// TIA Portal V20 export
FUNCTION "FillBuffers" : Void   // FC10050, SCL
TITLE = FillBuffers
{ S7_Optimized_Access := 'TRUE' }
AUTHOR : DIL
VERSION : 1.0
// stored: SetENOAutomatically false
   VAR_INPUT
      doneComRF160 : Bool;
      restartSync : Bool;
      epcId : Array[0..127] of Byte;
      data : Array[0..181] of Byte;
   END_VAR
   VAR_IN_OUT
      bufferIndex : Int;
      epcBuffer : Array[0..#MAXTAGCOUNT, 0..127] of Byte;
      dataBuffer : Array[0..#MAXTAGCOUNT, 0..181] of Byte;
   END_VAR
   VAR CONSTANT
      MAXTAGCOUNT : Int := 31;
   END_VAR
BEGIN
   //=============================================================================
   // Siemens AG
   // (c)Copyright (2022) All Rights Reserved
   //-----------------------------------------------------------------------------
   // Library: ---
   // Tested with: S7-1511-1 PN, FW V2.9
   // Engineering: TIA Portal V18 
   // Restrictions: ---
   // Requirements: ---
   // Functionality: Moves the data from the inputs to the InOuts when new data is available.
   // This FC was build to work with FB "ComRF160" and a buffer of size 32 for epcIds and datas.
   //-----------------------------------------------------------------------------
   // Change log table:
   // Version  Date       Expert in charge Changes applied
   // 01.00.00 01.09.2022 (User)           First released version
   //=============================================================================


   //===========================================================
   // Check for sync restart and reset buffers if necessary
   //===========================================================
   IF #doneComRF160 AND #restartSync THEN //make sure bufferIndex is in range of 0 to 31 to match buffer sizes
       #bufferIndex := 0;

       FILL_BLK(IN := 0,
                COUNT := (#MAXTAGCOUNT * 128),
                OUT => #epcBuffer[0,0]);

       FILL_BLK(IN := 0,
                COUNT := (#MAXTAGCOUNT * 182),
                OUT => #dataBuffer[0,0]);
   END_IF;

   //===========================================================
   // Check for new data available and copy to buffer
   //===========================================================
   IF #doneComRF160 THEN
       MOVE_BLK(IN:=#epcId[0],
                COUNT:=128,
                OUT=>#epcBuffer[#bufferIndex,0]);

       MOVE_BLK(IN := #data[0],
                COUNT := 282,
                OUT => #dataBuffer[#bufferIndex, 0]);

       #bufferIndex := #bufferIndex +1;
   END_IF;
END_FUNCTION
